{attribute addProperty BoxType "EL3773-0000-0018"}
{attribute addProperty Id "Sample_CountAT %I*UINT162"}
{attribute addProperty CRC "1190388509"}
{attribute addProperty SizeInBites "16"}
{attribute addProperty SizeInBytes "2"}
TYPE AI_Sample_Count_46F3E31D :
STRUCT
	{attribute addProperty Name "Sample_Count"}
	Sample_Count AT %I* : UINT;
END_STRUCT
END_TYPE

(* stored: Version 1.2.0.0, ProductVersion 3.1.4024.9
   DUT AI_Sample_Count_46F3E31D: Id {efd39f18-4065-4f6d-99eb-354888e66eef} *)
